FUNCTION_BLOCK FB_Cylinder_RetractedSensor EXTENDS FB_CylinderBase
VAR_INPUT
END_VAR
VAR_OUTPUT
END_VAR
VAR
	fbRetractedSensor			: FB_Sensor;
END_VAR

METHOD HardwareUpdate : BOOL
VAR_INPUT
END_VAR
fbSimExtend_TON();		//Call timer FB
fbSimRetract_TON();		//Call timer FB

GenerateFeedback(bExtend := bExtendCommand,
				 bRetract := bRetractCommand,
				 bExtended_Generated => bExtendedFeedback,
				 bRetracted_Generated => );
bRetractedFeedback := fbRetractedSensor.Active;
END_METHOD

END_FUNCTION_BLOCK

(* stored: Version 1.1.0.1, ProductVersion 3.1.4024.9
   POU FB_Cylinder_RetractedSensor: Id {5d0a56a3-8778-4147-a4dc-69578ffa4bd4}, SpecialFunc None
   Folder 01_SUPER_Overrides: Id {208af865-0f38-4b74-8b79-5dfe0815b948}
   Method HardwareUpdate: Id {15e214de-5b3c-4d17-ace1-412e71431e4f} *)
